Fanuc KAREL source: ks00041.KL

PROGRAM KS00041
%STACKSIZE=65535
%PRIORITY=65535
%NOLOCKGROUP
VAR
A : ARRAY[4] OF POSITION
B : ARRAY[4] OF POSITION
FLAG : BOOLEAN
N : INTEGER
STATUS : INTEGER
PN : STRING[80]
VN : STRING[80]
BEGIN
PN=''
VN='A'
-- UNRESOLVED_PC line 19 opcodes [27 22 22 2A 22 2A 22 22 AF] marker_code=27
END KS00041
